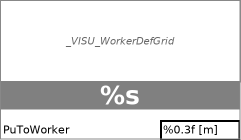
VISUALIZATION _VISU_WorkerDefGrid_Delete  // 241x140
VAR_IN_OUT
		m_Inst : FB_WorkerDefGrid_Delete;
END_VAR
    Frame (0,0 241x82)
        shows _VISU_WorkerDefGrid(m_Inst := m_Inst)
    Rectangle (0,80 240x30), "%s", text variable: m_Inst._name, colour toggle: m_Inst._pAttachedCt <> 0
    Rectangle (0,120 160x20), "PuToWorker"
    Rectangle (160,120 80x20), "%0.3f [m]", text variable: m_Inst._fWorkerToPu
        OnMouseDown: write the text variable via Default
END_VISUALIZATION

(* stored: Version 1.1.0.1, ProductVersion 3.1.4024.3
   Visu _VISU_WorkerDefGrid_Delete: Id {7c1799ac-baeb-4b99-a342-eddf0e1cf0f9} *)
